(* CoDeSys 2.3 export: TEMP.EXP *)

(* Global variable list: Global_Variables *)
VAR_GLOBAL
	posVelocity: REAL;
	posAcceleration: REAL;
	bMove1 AT %IX0.0: BOOL;
	bMove2 AT %IX0.1: BOOL;
	bMove3 AT %IX0.2: BOOL;
	bMove4 AT %IX0.3: BOOL;
	bInpos AT %QX0.0: BOOL;

END_VAR

(* POU PLC_PRG, FBD *)
PROGRAM PLC_PRG
VAR
	statusWord: WORD;
	fbPower: MC_Power;
	fbMove1: MC_MoveAbsolute;
	fbMove2: MC_MoveAbsolute;
	fbMove3: MC_MoveAbsolute;
	fbMove4: MC_MoveAbsolute;
	PosStatus: WORD;
	fbHome: MB_Home;
	bTeste: BOOL;
END_VAR
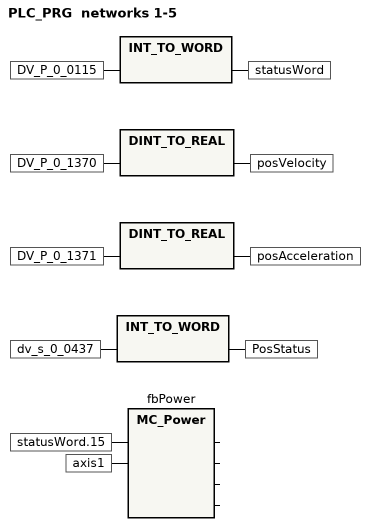
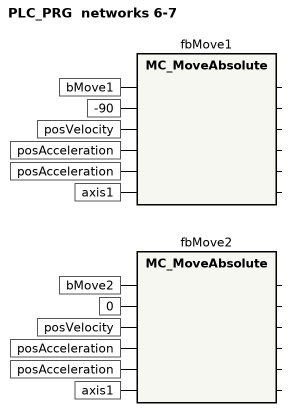
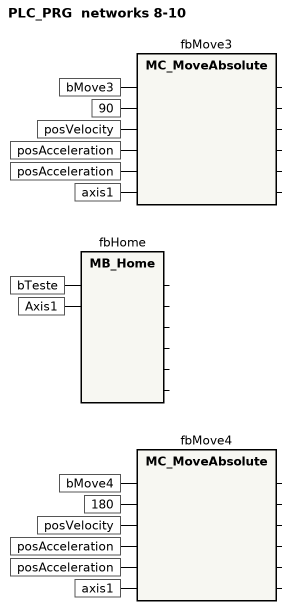
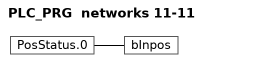
_FBD_ (* Function Block Diagram *)
NETWORK 1
	INT_TO_WORD(DV_P_0_0115) => statusWord
NETWORK 2
	DINT_TO_REAL(DV_P_0_1370) => posVelocity
NETWORK 3
	DINT_TO_REAL(DV_P_0_1371) => posAcceleration
NETWORK 4
	INT_TO_WORD(dv_s_0_0437) => PosStatus
NETWORK 5
	fbPower:MC_Power(statusWord.15, axis1)
NETWORK 6
	fbMove1:MC_MoveAbsolute(bMove1, -90, posVelocity, posAcceleration, posAcceleration, axis1)
NETWORK 7
	fbMove2:MC_MoveAbsolute(bMove2, 0, posVelocity, posAcceleration, posAcceleration, axis1)
NETWORK 8
	fbMove3:MC_MoveAbsolute(bMove3, 90, posVelocity, posAcceleration, posAcceleration, axis1)
NETWORK 9
	fbHome:MB_Home(bTeste, Axis1)
NETWORK 10
	fbMove4:MC_MoveAbsolute(bMove4, 180, posVelocity, posAcceleration, posAcceleration, axis1)
NETWORK 11
	PosStatus.0 => bInpos
_END_FBD_
(* the same logic as Structured Text *)
(* Network 1 *)
statusWord := INT_TO_WORD(DV_P_0_0115);
(* Network 2 *)
posVelocity := DINT_TO_REAL(DV_P_0_1370);
(* Network 3 *)
posAcceleration := DINT_TO_REAL(DV_P_0_1371);
(* Network 4 *)
PosStatus := INT_TO_WORD(dv_s_0_0437);
(* Network 5 *)
fbPower(statusWord.15, axis1);
(* Network 6 *)
fbMove1(bMove1, -90, posVelocity, posAcceleration, posAcceleration, axis1);
(* Network 7 *)
fbMove2(bMove2, 0, posVelocity, posAcceleration, posAcceleration, axis1);
(* Network 8 *)
fbMove3(bMove3, 90, posVelocity, posAcceleration, posAcceleration, axis1);
(* Network 9 *)
fbHome(bTeste, Axis1);
(* Network 10 *)
fbMove4(bMove4, 180, posVelocity, posAcceleration, posAcceleration, axis1);
(* Network 11 *)
bInpos := PosStatus.0;
END_PROGRAM
